(* Logix 5000 project; controller cal1615 1756-L62 rev 20.11; software revision 20.05; part 3 of 81 *)

ADD_ON_INSTRUCTION sys_ACS880_Outputs   (* revision 1.0 *)
// System AOI
// ACS880 Outputs
VAR_IN_OUT
   IO_vfd_outputs : AB:ETHERNET_MODULE_INT_24Bytes:O:0; {required}
   IO_vfd_data : vfd_data_ACS880; {required}   // VFD Data Object
END_VAR
VAR_INPUT
   IN_Gear_Reduction : REAL; {required}
   IN_Roll_Diameter : REAL; {required}
   IN_Speed_Setpoint : REAL; {required}
END_VAR
VAR_OUTPUT
   Out_Speed_Command : REAL; {access Read Only, visible}
   OUT_Speed_RPM : REAL; {access Read Only, visible}
END_VAR
VAR
   speed_hz : REAL;   // Speed Setpoint in Hz
   speed_pct : REAL;   // Motor Speed Percent
END_VAR

ROUTINE Logic   (* ladder *)
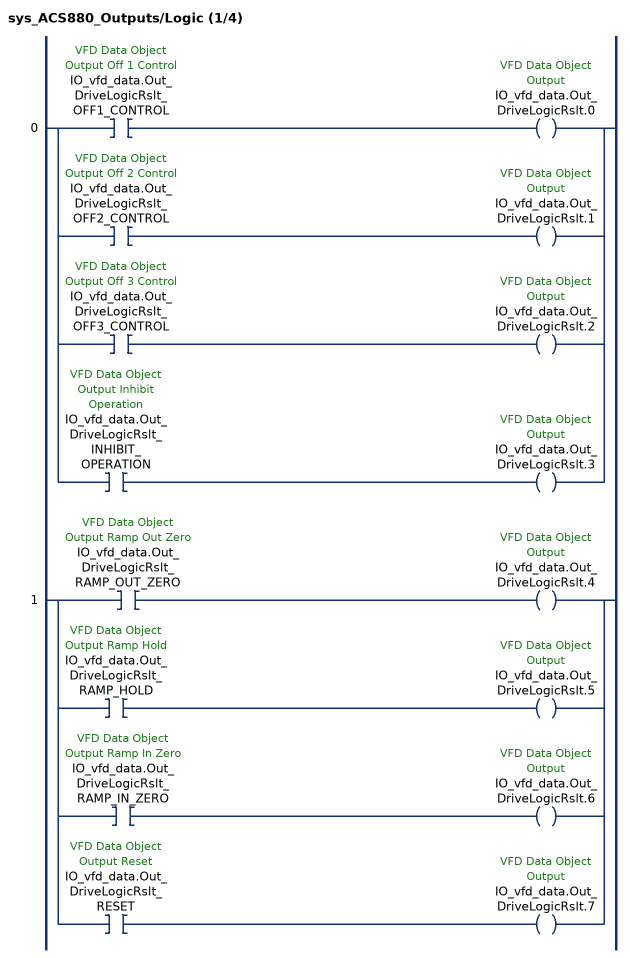
   0: [XIC(IO_vfd_data.Out_DriveLogicRslt_OFF1_CONTROL) OTE(IO_vfd_data.Out_DriveLogicRslt.0) ,XIC(IO_vfd_data.Out_DriveLogicRslt_OFF2_CONTROL) OTE(IO_vfd_data.Out_DriveLogicRslt.1) ,XIC(IO_vfd_data.Out_DriveLogicRslt_OFF3_CONTROL) OTE(IO_vfd_data.Out_DriveLogicRslt.2) ,XIC(IO_vfd_data.Out_DriveLogicRslt_INHIBIT_OPERATION) OTE(IO_vfd_data.Out_DriveLogicRslt.3) ];
   1: [XIC(IO_vfd_data.Out_DriveLogicRslt_RAMP_OUT_ZERO) OTE(IO_vfd_data.Out_DriveLogicRslt.4) ,XIC(IO_vfd_data.Out_DriveLogicRslt_RAMP_HOLD) OTE(IO_vfd_data.Out_DriveLogicRslt.5) ,XIC(IO_vfd_data.Out_DriveLogicRslt_RAMP_IN_ZERO) OTE(IO_vfd_data.Out_DriveLogicRslt.6) ,XIC(IO_vfd_data.Out_DriveLogicRslt_RESET) OTE(IO_vfd_data.Out_DriveLogicRslt.7) ];
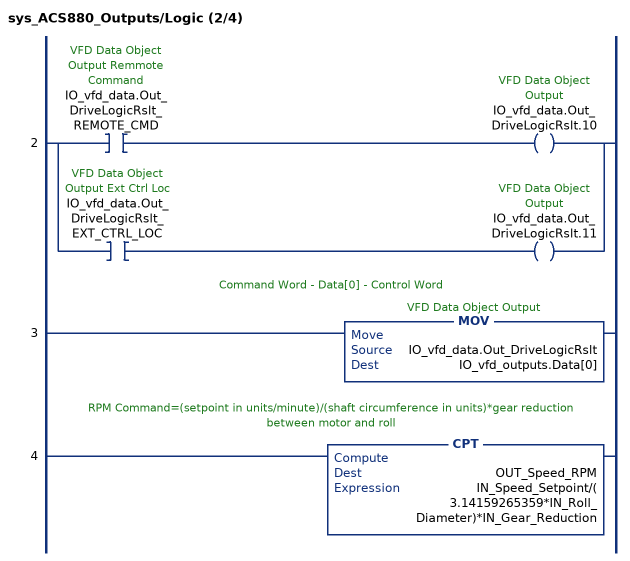
   2: [XIC(IO_vfd_data.Out_DriveLogicRslt_REMOTE_CMD) OTE(IO_vfd_data.Out_DriveLogicRslt.10) ,XIC(IO_vfd_data.Out_DriveLogicRslt_EXT_CTRL_LOC) OTE(IO_vfd_data.Out_DriveLogicRslt.11) ];
   // Command Word - Data[0] - Control Word
   3: MOV(IO_vfd_data.Out_DriveLogicRslt,IO_vfd_outputs.Data[0]);
   // RPM Command=(setpoint in units/minute)/(shaft circumference in units)*gear reduction between motor and roll
   4: CPT(OUT_Speed_RPM,IN_Speed_Setpoint/( 3.14159265359*IN_Roll_Diameter)*IN_Gear_Reduction);
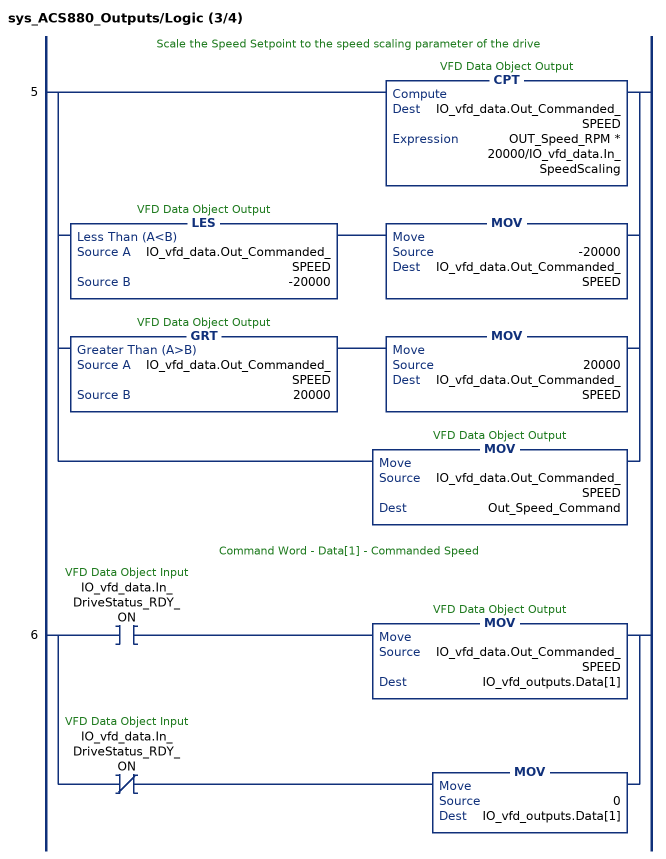
   // Scale the Speed Setpoint to the speed scaling parameter of the drive
   5: [CPT(IO_vfd_data.Out_Commanded_SPEED,OUT_Speed_RPM * 20000/IO_vfd_data.In_SpeedScaling) ,LES(IO_vfd_data.Out_Commanded_SPEED,-20000) MOV(-20000,IO_vfd_data.Out_Commanded_SPEED) ,GRT(IO_vfd_data.Out_Commanded_SPEED,20000) MOV(20000,IO_vfd_data.Out_Commanded_SPEED) ,MOV(IO_vfd_data.Out_Commanded_SPEED,Out_Speed_Command) ];
   // Command Word - Data[1] - Commanded Speed
   6: [XIC(IO_vfd_data.In_DriveStatus_RDY_ON) MOV(IO_vfd_data.Out_Commanded_SPEED,IO_vfd_outputs.Data[1]) ,XIO(IO_vfd_data.In_DriveStatus_RDY_ON) MOV(0,IO_vfd_outputs.Data[1]) ];
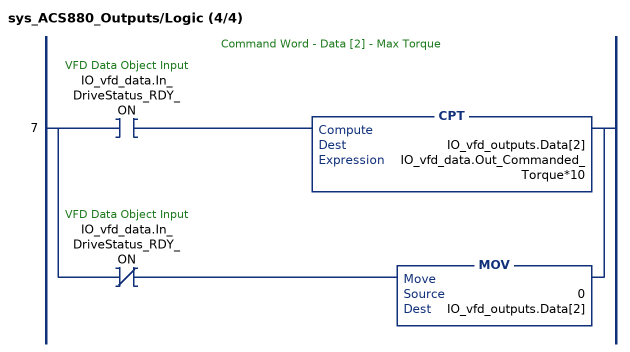
   // Command Word - Data [2] - Max Torque
   7: [XIC(IO_vfd_data.In_DriveStatus_RDY_ON) CPT(IO_vfd_outputs.Data[2],IO_vfd_data.Out_Commanded_Torque*10) ,XIO(IO_vfd_data.In_DriveStatus_RDY_ON) MOV(0,IO_vfd_outputs.Data[2]) ];
END_ROUTINE
END_ADD_ON_INSTRUCTION

ADD_ON_INSTRUCTION sys_ACS_FENA21   (* revision 1.0 *)
VAR_IN_OUT
   vfd_abb_data : vfd_data_ACS880; {required}
END_VAR
VAR_INPUT
   IN_START : BOOL; {required}
   IN_GLOBAL_RESET : BOOL; {required}
   IN_DRIVE_PERMISSIVE : BOOL; {required}
END_VAR
VAR_OUTPUT
   OUT_FAULT : BOOL; {access Read Only, visible}
   OUT_ALARM : BOOL; {access Read Only, visible}
   OUT_ENABLED : BOOL; {access Read Only, visible}
   DRIVE_NOT_READY_FAULT : BOOL; {access Read Only}
END_VAR

ROUTINE Logic   (* ladder *)
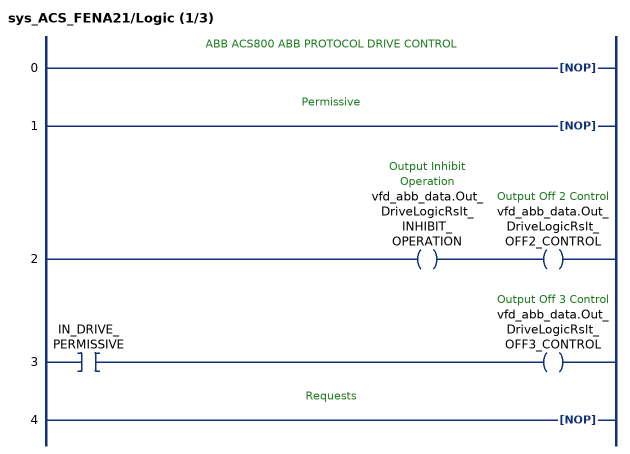
   // ABB ACS800 ABB PROTOCOL DRIVE CONTROL
   0: NOP();
   // Permissive
   1: NOP();
   2: OTE(vfd_abb_data.Out_DriveLogicRslt_INHIBIT_OPERATION)OTE(vfd_abb_data.Out_DriveLogicRslt_OFF2_CONTROL);
   3: XIC(IN_DRIVE_PERMISSIVE)OTE(vfd_abb_data.Out_DriveLogicRslt_OFF3_CONTROL);
   // Requests
   4: NOP();
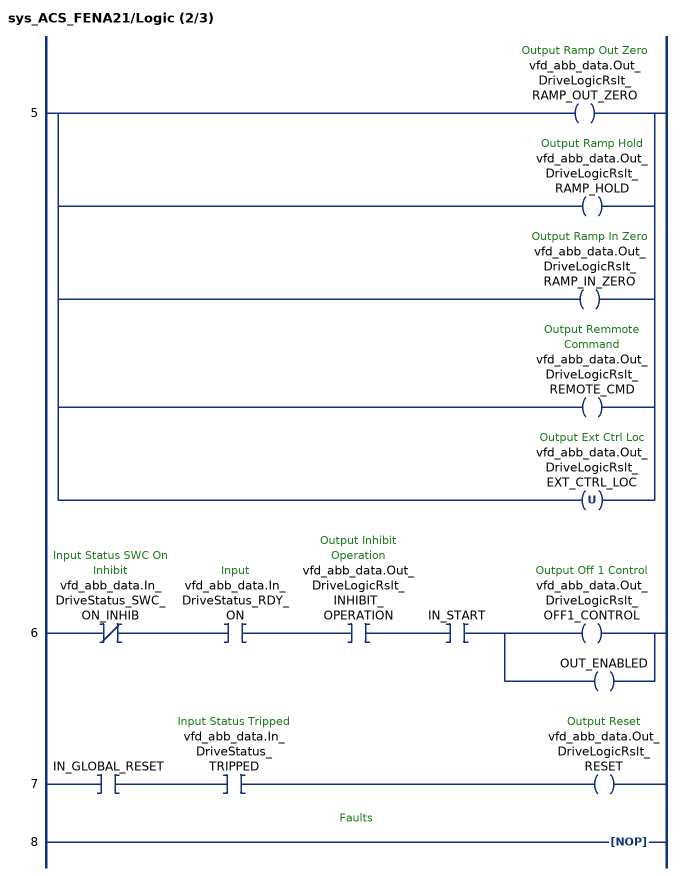
   5: [OTE(vfd_abb_data.Out_DriveLogicRslt_RAMP_OUT_ZERO) ,OTE(vfd_abb_data.Out_DriveLogicRslt_RAMP_HOLD) ,OTE(vfd_abb_data.Out_DriveLogicRslt_RAMP_IN_ZERO) ,OTE(vfd_abb_data.Out_DriveLogicRslt_REMOTE_CMD) ,OTU(vfd_abb_data.Out_DriveLogicRslt_EXT_CTRL_LOC) ];
   6: XIO(vfd_abb_data.In_DriveStatus_SWC_ON_INHIB)XIC(vfd_abb_data.In_DriveStatus_RDY_ON)XIC(vfd_abb_data.Out_DriveLogicRslt_INHIBIT_OPERATION)XIC(IN_START)[OTE(vfd_abb_data.Out_DriveLogicRslt_OFF1_CONTROL) ,OTE(OUT_ENABLED) ];
   7: XIC(IN_GLOBAL_RESET)XIC(vfd_abb_data.In_DriveStatus_TRIPPED)OTE(vfd_abb_data.Out_DriveLogicRslt_RESET);
   // Faults
   8: NOP();
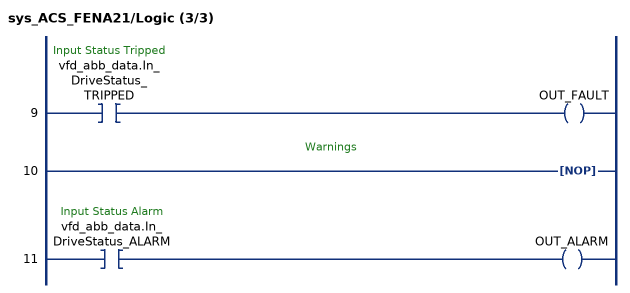
   9: XIC(vfd_abb_data.In_DriveStatus_TRIPPED)OTE(OUT_FAULT);
   // Warnings
   10: NOP();
   11: XIC(vfd_abb_data.In_DriveStatus_ALARM)OTE(OUT_ALARM);
END_ROUTINE
END_ADD_ON_INSTRUCTION

ADD_ON_INSTRUCTION SYS_ENC   (* revision 1.0 *)
VAR_INPUT
   IN_State : DINT; {required}
END_VAR
VAR_OUTPUT
   OUT_Status : DINT; {access Read Only, required}
END_VAR

ROUTINE Logic   (* ladder *)
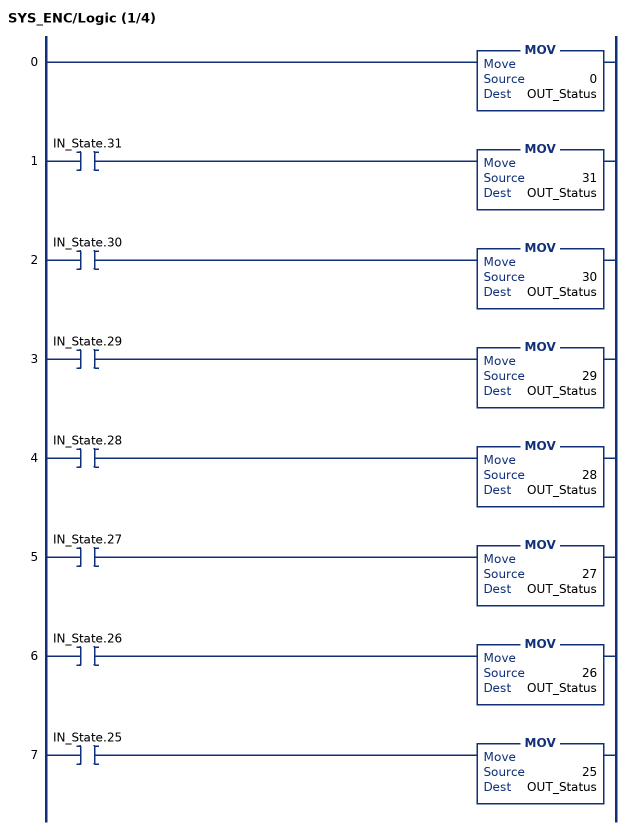
   0: MOV(0,OUT_Status);
   1: XIC(IN_State.31)MOV(31,OUT_Status);
   2: XIC(IN_State.30)MOV(30,OUT_Status);
   3: XIC(IN_State.29)MOV(29,OUT_Status);
   4: XIC(IN_State.28)MOV(28,OUT_Status);
   5: XIC(IN_State.27)MOV(27,OUT_Status);
   6: XIC(IN_State.26)MOV(26,OUT_Status);
   7: XIC(IN_State.25)MOV(25,OUT_Status);
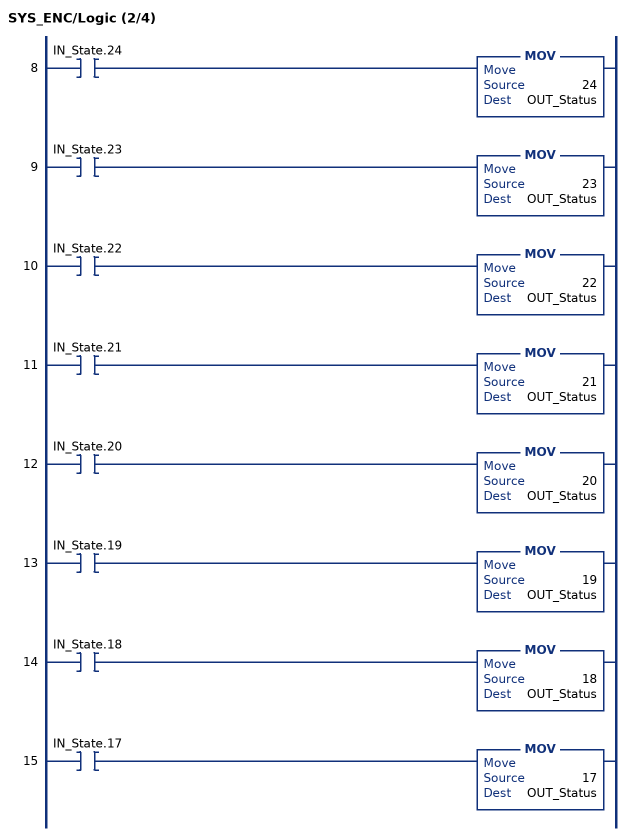
   8: XIC(IN_State.24)MOV(24,OUT_Status);
   9: XIC(IN_State.23)MOV(23,OUT_Status);
   10: XIC(IN_State.22)MOV(22,OUT_Status);
   11: XIC(IN_State.21)MOV(21,OUT_Status);
   12: XIC(IN_State.20)MOV(20,OUT_Status);
   13: XIC(IN_State.19)MOV(19,OUT_Status);
   14: XIC(IN_State.18)MOV(18,OUT_Status);
   15: XIC(IN_State.17)MOV(17,OUT_Status);
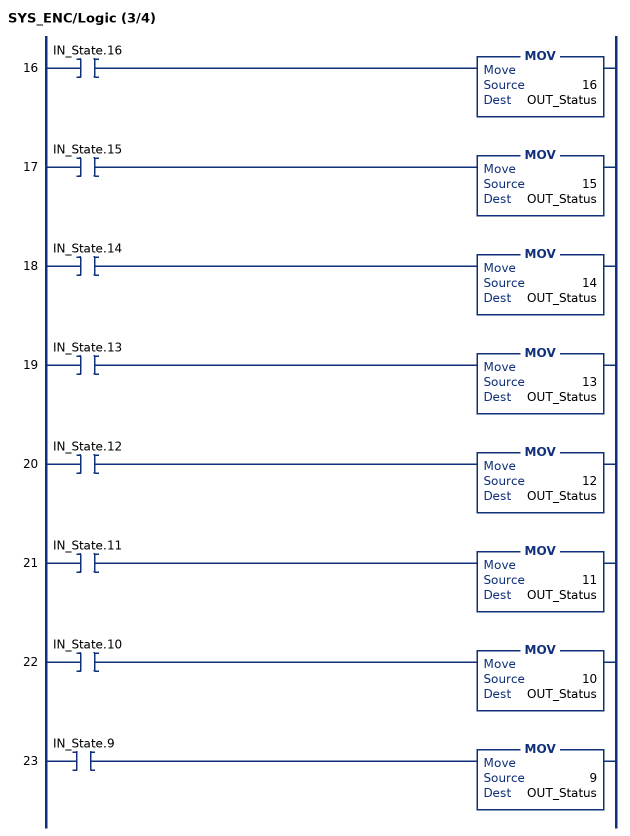
   16: XIC(IN_State.16)MOV(16,OUT_Status);
   17: XIC(IN_State.15)MOV(15,OUT_Status);
   18: XIC(IN_State.14)MOV(14,OUT_Status);
   19: XIC(IN_State.13)MOV(13,OUT_Status);
   20: XIC(IN_State.12)MOV(12,OUT_Status);
   21: XIC(IN_State.11)MOV(11,OUT_Status);
   22: XIC(IN_State.10)MOV(10,OUT_Status);
   23: XIC(IN_State.9)MOV(9,OUT_Status);
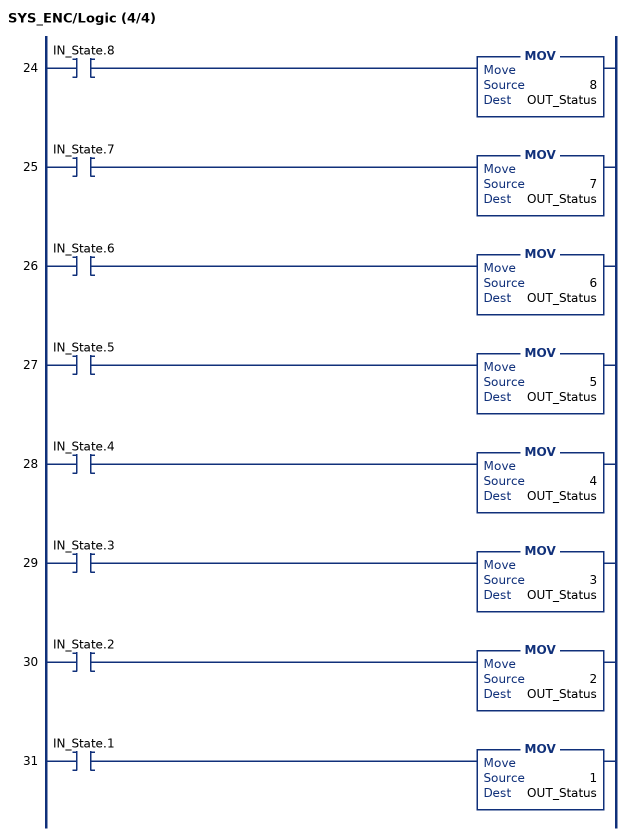
   24: XIC(IN_State.8)MOV(8,OUT_Status);
   25: XIC(IN_State.7)MOV(7,OUT_Status);
   26: XIC(IN_State.6)MOV(6,OUT_Status);
   27: XIC(IN_State.5)MOV(5,OUT_Status);
   28: XIC(IN_State.4)MOV(4,OUT_Status);
   29: XIC(IN_State.3)MOV(3,OUT_Status);
   30: XIC(IN_State.2)MOV(2,OUT_Status);
   31: XIC(IN_State.1)MOV(1,OUT_Status);
END_ROUTINE
END_ADD_ON_INSTRUCTION

ADD_ON_INSTRUCTION SYS_ENC_WITH_ZERO_BIT   (* revision 1.0 *)
VAR_INPUT
   IN_State : DINT; {required}
END_VAR
VAR_OUTPUT
   OUT_Status : DINT; {access Read Only, required}
END_VAR

ROUTINE Logic   (* ladder *)
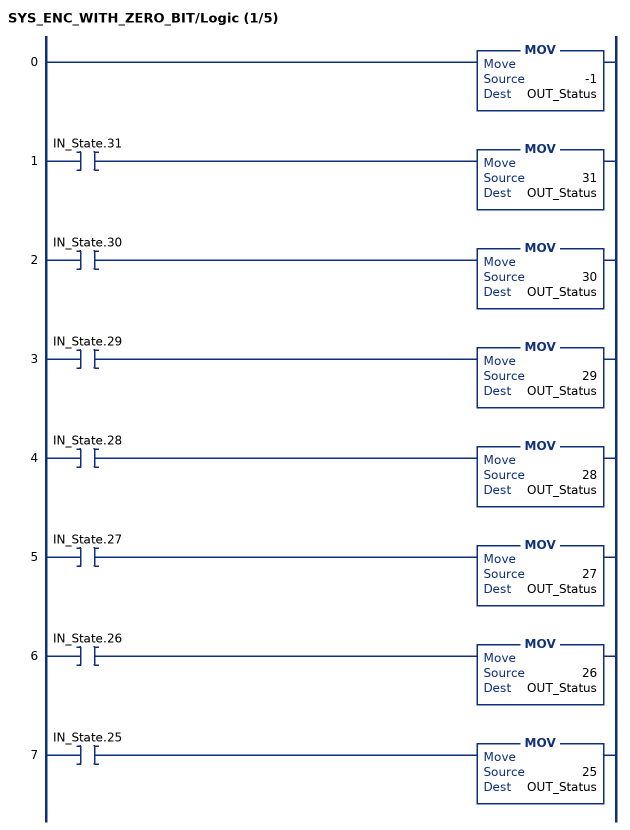
   0: MOV(-1,OUT_Status);
   1: XIC(IN_State.31)MOV(31,OUT_Status);
   2: XIC(IN_State.30)MOV(30,OUT_Status);
   3: XIC(IN_State.29)MOV(29,OUT_Status);
   4: XIC(IN_State.28)MOV(28,OUT_Status);
   5: XIC(IN_State.27)MOV(27,OUT_Status);
   6: XIC(IN_State.26)MOV(26,OUT_Status);
   7: XIC(IN_State.25)MOV(25,OUT_Status);
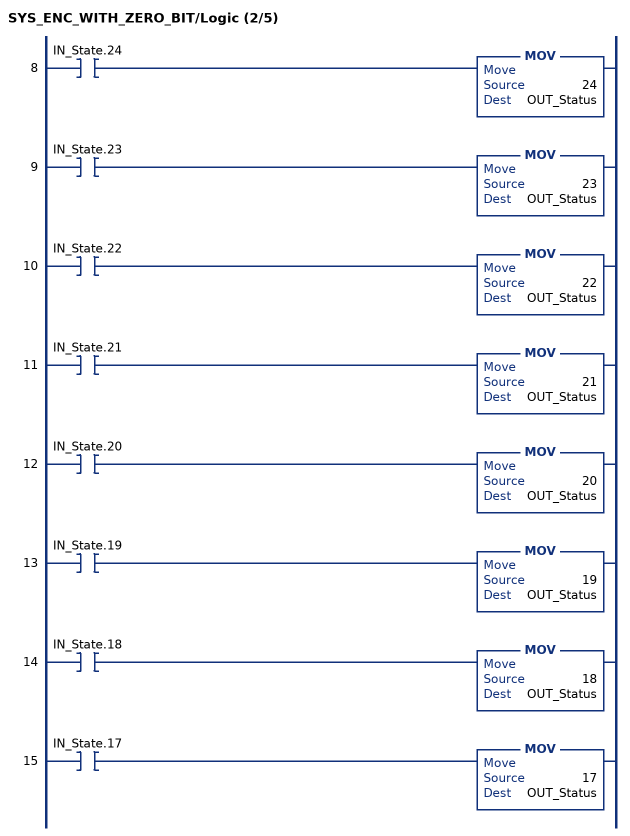
   8: XIC(IN_State.24)MOV(24,OUT_Status);
   9: XIC(IN_State.23)MOV(23,OUT_Status);
   10: XIC(IN_State.22)MOV(22,OUT_Status);
   11: XIC(IN_State.21)MOV(21,OUT_Status);
   12: XIC(IN_State.20)MOV(20,OUT_Status);
   13: XIC(IN_State.19)MOV(19,OUT_Status);
   14: XIC(IN_State.18)MOV(18,OUT_Status);
   15: XIC(IN_State.17)MOV(17,OUT_Status);
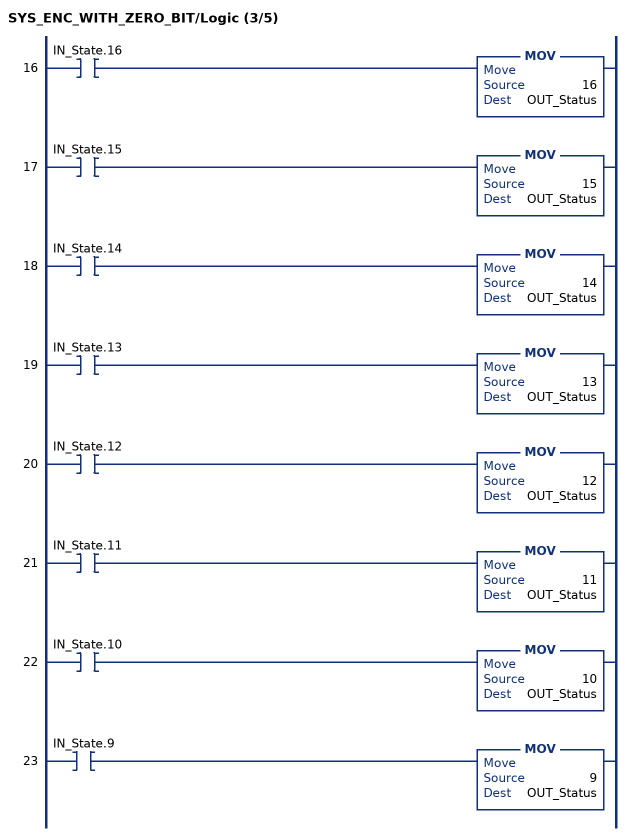
   16: XIC(IN_State.16)MOV(16,OUT_Status);
   17: XIC(IN_State.15)MOV(15,OUT_Status);
   18: XIC(IN_State.14)MOV(14,OUT_Status);
   19: XIC(IN_State.13)MOV(13,OUT_Status);
   20: XIC(IN_State.12)MOV(12,OUT_Status);
   21: XIC(IN_State.11)MOV(11,OUT_Status);
   22: XIC(IN_State.10)MOV(10,OUT_Status);
   23: XIC(IN_State.9)MOV(9,OUT_Status);
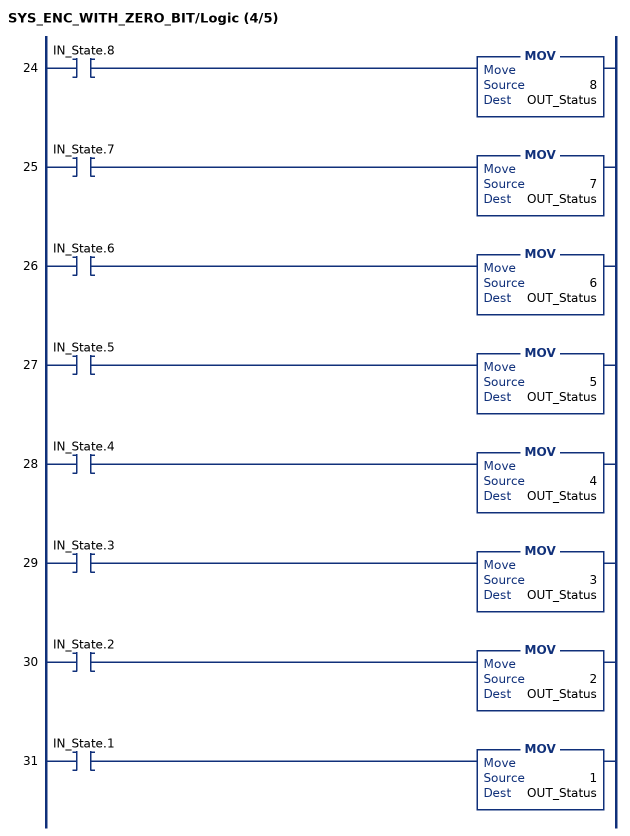
   24: XIC(IN_State.8)MOV(8,OUT_Status);
   25: XIC(IN_State.7)MOV(7,OUT_Status);
   26: XIC(IN_State.6)MOV(6,OUT_Status);
   27: XIC(IN_State.5)MOV(5,OUT_Status);
   28: XIC(IN_State.4)MOV(4,OUT_Status);
   29: XIC(IN_State.3)MOV(3,OUT_Status);
   30: XIC(IN_State.2)MOV(2,OUT_Status);
   31: XIC(IN_State.1)MOV(1,OUT_Status);
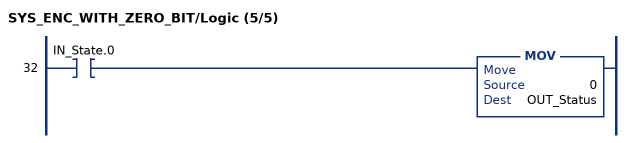
   32: XIC(IN_State.0)MOV(0,OUT_Status);
END_ROUTINE
END_ADD_ON_INSTRUCTION

ADD_ON_INSTRUCTION sys_Filter   (* revision 1.0, vendor Rockwell Automation *)
// System
// Filter
VAR_INPUT
   filter : REAL; {required}
   In_real : REAL; {required}
END_VAR
VAR_OUTPUT
   Out_Real : REAL; {access Read Only, required}
END_VAR
VAR
   LDL2_01 : LEAD_LAG_SEC_ORDER := (ZetaLag := 0.05, Order := 1, RTSTime := 1);
   LDL2_02 : LEAD_LAG_SEC_ORDER := (ZetaLag := 0.05, Order := 1, RTSTime := 1);
   __l01DD61F468DFC2B0 : REAL;
   __l01DD1CDF68DFBBC6 : REAL;
END_VAR

ROUTINE Logic   (* function block diagram *)
   SHEET 1
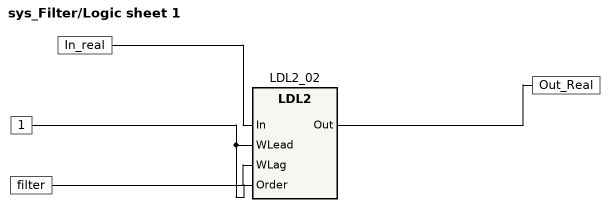
   LDL2_02 : LDL2(In := In_real, WLead := 1, WLag := filter, Order := 1);
   Out_Real := LDL2_02.Out;
END_ROUTINE
END_ADD_ON_INSTRUCTION

ADD_ON_INSTRUCTION sys_Limit_Clamp   (* revision 1.0, vendor Rockwell Automation *)
// System Block
// Limit Clamp
VAR_INPUT
   max : REAL; {required}
   min : REAL; {required}
END_VAR
VAR_IN_OUT
   variable : REAL; {required}
END_VAR

ROUTINE Logic   (* ladder *)
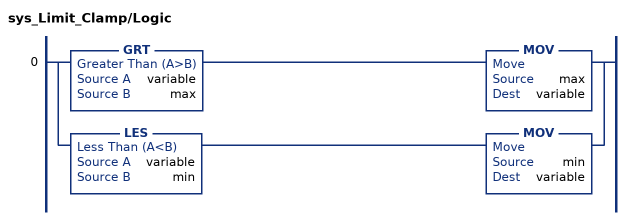
   0: [GRT(variable,max) MOV(max,variable) ,LES(variable,min) MOV(min,variable) ];
END_ROUTINE
END_ADD_ON_INSTRUCTION
